// TwinCAT 3 PLC project PLC
// ProgramVersion: 3.1.4022.7
// libraries:
//   Tc2_Standard, * (Beckhoff Automation GmbH)
//   Tc2_System, * (Beckhoff Automation GmbH)
//   Tc2_Utilities, * (Beckhoff Automation GmbH)
//   Tc3_Module, * (Beckhoff Automation GmbH)
//   TcUnit, * (www.tcunit.org)
// project tree:
//   Behavioral Patterns/Command/ I_Command.TcIO, NoCommand.TcPOU
//   Behavioral Patterns/Observer/ Class Diagram Observer.TcCD (not stored), Observable.TcPOU, I_Observable.TcIO, I_Observer.TcIO
//   Behavioral Patterns/Singleton/ I_Singleton.TcIO, Singleton.TcPOU, MySingleton.TcPOU
//   Test/Behavioral Patterns/Singleton/ SingletonPatternTest.TcPOU
//   UseCase/Behavioral Patterns/Command/Clients %28Receivers%29/ Gate.TcPOU (not stored), Light.TcPOU (not stored)
//   UseCase/Behavioral Patterns/Command/Commands/ I_OffCommand.TcIO, I_CloseCommand.TcIO, I_OnCommand.TcIO, I_OpenCommand.TcIO, OffCommand.TcPOU, CloseCommand.TcPOU, OnCommand.TcPOU, OpenCommand.TcPOU
//   UseCase/Behavioral Patterns/Command/Invokers/ Tp10.TcPOU
//   UseCase/Behavioral Patterns/Command/ P_CommandPattern.TcPOU
//   UseCase/Behavioral Patterns/Decorator/ P_Decorator.TcPOU
//   UseCase/Behavioral Patterns/Decorator/StringBuilder/ StringBuilder.TcPOU
//   UseCase/Behavioral Patterns/Singleton/ P_Singleton.TcPOU
//   UseCase/Behavioral Patterns/Singleton/SingletonByProxy1/ P_SingletonByProxy.TcPOU, ProxyToSingleton.TcPOU, Proxy_Interface.TcIO, RealSingleton.TcPOU
//   UseCase/Behavioral Patterns/Singleton/SingletonByProxy/ I_MessageLogger.TcIO, MessageLogger.TcPOU, MessageLoggerSingleton.TcPOU
//   _Interfaces/ I_CyclicCall.TcIO
//   / MAIN.TcPOU, Param.TcGVL, PlcTask.TcTTO
//   Test/Behavioral Patterns/Observer/ ObserverPatternTest.TcPOU
//   Test/ P_TEST.TcPOU
//   UseCase/Behavioral Patterns/Observer/ EventPublisherWithInheritance.TcPOU, EventPublisherWithoutInheritance.TcPOU, FB_EventSubscriber.TcPOU, FB_EventSubscriber2.TcPOU, I_EventPublisher.TcIO, P_ObserverPattern.TcPOU, _Class Diagram Observer Use Case.TcCD (not stored)
//   UseCase/ P_USE_CASES.TcPOU
// real-time tasks:
//   TASK PlcTask: cycle T#10ms, priority 20, ADS port 350

CONFIGURATION PLC
    RESOURCE PLC ON TwinCAT3
        TASK PlcTask(INTERVAL := T#10ms, PRIORITY := 20);
        PROGRAM MAIN WITH PlcTask : MAIN;
    END_RESOURCE
END_CONFIGURATION

// ---- Param.TcGVL
{attribute 'qualified_only'}
VAR_GLOBAL CONSTANT
	MaxObservers 	: INT := 5;	
END_VAR

// ---- Behavioral Patterns/Command/I_Command.TcIO
INTERFACE I_Command

METHOD Execute
VAR_INPUT
END_VAR
END_METHOD

END_INTERFACE

// ---- Behavioral Patterns/Observer/I_Observable.TcIO
INTERFACE I_Observable

METHOD Attach : bool
VAR_INPUT
	observer			: I_Observer;
END_VAR
END_METHOD

METHOD Detach : BOOL
VAR_INPUT
	observer			: I_Observer;
END_VAR
END_METHOD

END_INTERFACE

// ---- Behavioral Patterns/Observer/I_Observer.TcIO
INTERFACE I_Observer

METHOD Update : BOOL
VAR_INPUT
END_VAR
END_METHOD

END_INTERFACE

// ---- Behavioral Patterns/Singleton/I_Singleton.TcIO
INTERFACE I_Singleton

METHOD Message : String
VAR_INPUT
END_VAR
END_METHOD

END_INTERFACE

// ---- UseCase/Behavioral Patterns/Command/Commands/I_OffCommand.TcIO
INTERFACE I_OffCommand

PROPERTY IsOff : Bool
GET
END_GET
END_PROPERTY

METHOD Off
END_METHOD

END_INTERFACE

// ---- UseCase/Behavioral Patterns/Command/Commands/I_CloseCommand.TcIO
INTERFACE I_CloseCommand

METHOD Close
END_METHOD

PROPERTY IsClosed : Bool
GET
END_GET
END_PROPERTY

END_INTERFACE

// ---- UseCase/Behavioral Patterns/Command/Commands/I_OnCommand.TcIO
INTERFACE I_OnCommand

PROPERTY IsOn : Bool
GET
END_GET
END_PROPERTY

METHOD On
END_METHOD

END_INTERFACE

// ---- UseCase/Behavioral Patterns/Command/Commands/I_OpenCommand.TcIO
INTERFACE I_OpenCommand

PROPERTY IsOpen : Bool
GET
END_GET
END_PROPERTY

METHOD Open
END_METHOD

END_INTERFACE

// ---- UseCase/Behavioral Patterns/Singleton/SingletonByProxy1/Proxy_Interface.TcIO
INTERFACE Proxy_Interface

///Illustrative method of the pattern
METHOD Set_Background
VAR_INPUT
	///HEX value to be set as background color
	newBackground: DWORD;
END_VAR
END_METHOD

END_INTERFACE

// ---- UseCase/Behavioral Patterns/Singleton/SingletonByProxy/I_MessageLogger.TcIO
INTERFACE I_MessageLogger

METHOD LogMessage : String
VAR_INPUT
	Message			: STRING;
END_VAR
END_METHOD

PROPERTY message : string
GET
END_GET
END_PROPERTY

END_INTERFACE

// ---- _Interfaces/I_CyclicCall.TcIO
INTERFACE I_CyclicCall

METHOD CyclicCall
END_METHOD

END_INTERFACE

// ---- UseCase/Behavioral Patterns/Observer/I_EventPublisher.TcIO
INTERFACE I_EventPublisher EXTENDS I_Observable

PROPERTY Event : int
GET
END_GET
END_PROPERTY

END_INTERFACE

// ---- MAIN.TcPOU
PROGRAM MAIN
VAR
// *************** ROUTER
	// router info (memory consumption)
	fbGetRouterStatusInfo 	: FB_GetRouterStatusInfo;
	stTCRouterStatusInfo	: ST_TCRouterStatusInfo;
	memAvailable			: DWORD;
END_VAR

// TcUnit tests
P_TEST();

// Use cases implementations
P_USE_CASES();

// *************** ROUTER INFO
// router status
fbGetRouterStatusInfo(
	sNetId:= , 
	bExecute:= NOT fbGetRouterStatusInfo.bBusy, 
	tTimeout:= , 
	bBusy=> , 
	bError=> , 
	nErrID=> , 
	info=> stTCRouterStatusInfo
	);
IF stTCRouterStatusInfo.maxMemAvail	> 0 THEN
	memAvailable := stTCRouterStatusInfo.maxMemAvail;
END_IF

END_PROGRAM

// ---- Test/P_TEST.TcPOU
PROGRAM P_TEST
VAR
	fbObserver_Pattern_Test					: ObserverPatternTest;
	fbSingleton_Pattern_Test				: SingletonPatternTest;
END_VAR

tcUnit.RUN();

END_PROGRAM

// ---- Test/Behavioral Patterns/Observer/ObserverPatternTest.TcPOU
FUNCTION_BLOCK ObserverPatternTest EXTENDS tcUnit.FB_TestSuite
VAR
	// Unit test use the implementation of the use case so both 
	// base blocks and use case blocks are tested at once
	eventPublisher					: EventPublisherWithInheritance;
	//eventSubscriber					: ARRAY[1..param.MaxObservers+1] OF FB_EventSubscriber[(eventPublisher),(eventPublisher),(0),(0),(0),(0)];	// Max + 1 for unit test	// Pass the interface reference to the instances is not possible?	
	eventSubscriber					: ARRAY[1..param.MaxObservers+1] OF FB_EventSubscriber(0);	// Max + 1 for unit test	// Pass the interface reference to the instances is not possible?	
END_VAR

ObservableAttachesAnObserver();
ObservableAttachesASecondObserver();
ObservableAttachesTooMuchObservers();
ObserverFetchesCorrectData();

METHOD ObservableAttachesAnObserver
TEST('ObservableAttachesAnObserver');

// pass observee to subscriber
eventSubscriber[1].ChangePublisher(eventPublisher);

// First loop attaches the observer to the observee 
eventSubscriber[1].CyclicCall();

// One subscriber should be attached
AssertEquals_INT(
	Expected	:= 1, 
	Actual		:= eventPublisher.NoOfAttachedObservers, 
	Message 	:= 'Attaching a subscriber failed'
	);
	
TEST_FINISHED();
END_METHOD

METHOD ObservableAttachesASecondObserver
TEST('ObservableAttachesASecondObserver');

// pass observee to subscriber
eventSubscriber[2].ChangePublisher(eventPublisher);

// First loop attaches another observer to the observee 
eventSubscriber[2].CyclicCall();

// One extra subscriber should be attached
AssertEquals_INT(
	Expected	:= 2, 
	Actual		:= eventPublisher.NoOfAttachedObservers, 
	Message 	:= 'Attaching a second subscriber failed'
	);
	
TEST_FINISHED();
END_METHOD

METHOD ObservableAttachesTooMuchObservers
VAR
	i						: INT;
END_VAR
TEST('ObservableAttachesTooMuchObservers');

// First loop attaches another observer to the observee 
FOR i := 3 TO Param.MaxObservers + 1 DO
	// pass observee to subscriber
	eventSubscriber[i].ChangePublisher(eventPublisher);
	eventSubscriber[i].CyclicCall();
END_FOR
	
// Max no of subscribers should be attached
AssertEquals_INT(
	Expected	:= Param.MaxObservers, 
	Actual		:= eventPublisher.NoOfAttachedObservers, 
	Message 	:= 'Too many subscribers were registered'
	);
	
TEST_FINISHED();
END_METHOD

// Tests the complete observer pattern flow
METHOD ObserverFetchesCorrectData
VAR
	message					: T_MaxString;
	fbFormatString			: FB_FormatString;
	i: INT;
END_VAR
TEST('ObserverFetchesCorrectData');

// Change the event in the publisher (in the example it is an INT) 
eventPublisher.ChangeEvent := eventPublisher.Event + 1;
eventPublisher.CyclicCall();

FOR i := 1 TO Param.MaxObservers DO
	fbFormatString(sFormat:= 'Observer %d did not receive the correct data', arg1:= F_INT(i), sOut=> message);
	AssertEquals_INT(1 , eventSubscriber[i].event, message);
END_FOR

TEST_FINISHED();
END_METHOD

END_FUNCTION_BLOCK

// ---- UseCase/Behavioral Patterns/Observer/EventPublisherWithInheritance.TcPOU
{attribute 'no_explicit_call' := 'FB_EventPublisher is a CLASS and must be accessed using methods or properties'}
FUNCTION_BLOCK EventPublisherWithInheritance EXTENDS Observable IMPLEMENTS I_CyclicCall, I_EventPublisher
VAR
	_event							: INT;
	eventPrev						: INT;
END_VAR


// The body of a class must not be used for code.  
// Cyclic code should be called from a method if needed.

PROPERTY PUBLIC ChangeEvent : int
SET
// IMPLEMENTED ONLY FOR TESTING PURPOSES
VAR
END_VAR
_event := changeEvent;
END_SET
END_PROPERTY

METHOD CyclicCall
IF eventPrev <> _event 			THEN
	notify();
	eventPrev := _event;
END_IF
END_METHOD

// IMPLEMENTED ONLY FOR TESTING PURPOSES
PROPERTY Event : int
GET
event := _event;
END_GET
END_PROPERTY

END_FUNCTION_BLOCK

// ---- Behavioral Patterns/Observer/Observable.TcPOU
{attribute 'no_explicit_call' := 'Observable is a CLASS and must be accessed using methods or properties'}
FUNCTION_BLOCK Observable IMPLEMENTS I_Observable
VAR
	verbose							: BOOL := TRUE;
	// Make sure the list of references to subscribers is updated after online change 
	observers						: ARRAY[1..param.MaxObservers] OF I_Observer;
END_VAR


// The body of a class must not be used for code.  
// Cyclic code should be called from a method if needed.

METHOD Attach : BOOL
VAR_INPUT
	observer			: I_Observer;
END_VAR
VAR
	i					: INT;
END_VAR
(* default *)
attach := FALSE;

(* loop if the subscriber is already registered *)
FOR i := 1 TO param.MaxObservers DO
	IF observers[i] = observer 	THEN
		observer.update();
		attach := TRUE;
		RETURN;
	END_IF
END_FOR

(* loop for first free position if not yet attached *)
FOR i := 1 TO param.MaxObservers DO
	IF observers[i] = 0 	THEN
		observers[i] := observer;
		message('Observer registered');
		observer.update();
		attach := TRUE;
		EXIT;
	END_IF
END_FOR
END_METHOD

METHOD Detach : BOOL
VAR_INPUT
	observer			: I_Observer;
END_VAR
VAR
	i					: INT;
END_VAR
(* default *)
detach := FALSE;

(* loop if the subscriber is already registered *)
FOR i := 1 TO param.MaxObservers DO
	IF observers[i] = observer 	THEN
		observers[i] := 0;
		message('Observer deregistered');
		detach := TRUE;
		RETURN;
	END_IF
END_FOR
END_METHOD

{attribute 'call_after_online_change_slot' := '0'}
METHOD PRIVATE fbreinit
(*	!!!!!!!!!!!!!!!!!!!!!!!!!!!!!!!!!
   	THIS METHOD is force called after every online change 
   	!= the fb_reinit system call that will be called after the instance of the concerned function block has been copied 
 	(during an online change after modifications in the function block declaration)

	This is necessary since both observer en observee have references to one other
	!!!!!!!!!!!!!!!!!!!!!!!!!!!!!!!!!	*) 
VAR
	i					: INT;
END_VAR
(* loop if the subscriber is already registered *)
FOR i := 1 TO param.MaxObservers DO
	observers[i] := 0;
END_FOR
breinit:=NOT breinit; // flip the test marker
END_METHOD

METHOD PRIVATE Message : BOOL
VAR_INPUT
	strArg						: STRING;
END_VAR
// Log message
IF verbose  THEN
	ADSLOGSTR(
		msgCtrlMask := ADSLOG_MSGTYPE_HINT OR ADSLOG_MSGTYPE_LOG, // ADSLOG_MSGTYPE_ERROR OR ADSLOG_MSGTYPE_LOG, 
		msgFmtStr 	:= '%s',
		strArg 		:= strArg
		);
END_IF
END_METHOD

PROPERTY NoOfAttachedObservers : int
GET
VAR
	i							: INT;
END_VAR
// In stead of using an internal counter that could fail
// run through the array of attached observers
(* loop for first free position if not yet attached *)
NoOfAttachedObservers := 0;
FOR i := 1 TO param.MaxObservers DO
	IF observers[i] <> 0 	THEN
		NoOfAttachedObservers := NoOfAttachedObservers + 1;
	END_IF
END_FOR
END_GET
END_PROPERTY

METHOD Notify : BOOL
VAR
	i			: INT;
END_VAR
(* default *)
notify := FALSE;

(* loop if the subscriber is already registered *)
FOR i := 1 TO param.MaxObservers DO
	IF observers[i] <> 0 	THEN
		observers[i].update();
	END_IF
END_FOR
END_METHOD

END_FUNCTION_BLOCK

// ---- UseCase/Behavioral Patterns/Observer/FB_EventSubscriber.TcPOU
{attribute 'no_explicit_call' := 'FB_EventSubscriber is a CLASS and must be accessed using methods or properties'}
FUNCTION_BLOCK FB_EventSubscriber IMPLEMENTS I_CyclicCall, I_Observer
VAR	
	_eventPublisher					: I_EventPublisher;
	_event							: INT;
	
	verbose							: BOOL := TRUE;

	// Register after online change 
	registeredAtPublisher			: BOOL;	
	
	
	arr				: ARRAY[0..100] OF BOOL;
END_VAR


// The body of a class must not be used for code.  
// Cyclic code should be called from a method if needed.

METHOD ChangePublisher
VAR_INPUT
	eventPublisher					: I_EventPublisher;
END_VAR
_eventPublisher := eventPublisher;
END_METHOD

METHOD CyclicCall
// Did we already register in the publisher?
IF NOT registeredAtPublisher	THEN
	registeredAtPublisher := _eventPublisher.attach(THIS^);
END_IF
END_METHOD

// IMPLEMENTED ONLY FOR TESTING PURPOSES
PROPERTY Event : int
GET
event := _event;
END_GET
END_PROPERTY

METHOD FB_init : BOOL
VAR_INPUT
	bInitRetains	 				: BOOL; // if TRUE, the retain variables are initialized (warm start / cold start)
	bInCopyCode 					: BOOL;  // if TRUE, the instance afterwards gets moved into the copy code (online change)
	EventPublisher					: I_EventPublisher;
END_VAR
_eventPublisher := eventPublisher;
END_METHOD

{attribute 'call_after_online_change_slot' := '0'}
METHOD PRIVATE fbreinit

(*	!!!!!!!!!!!!!!!!!!!!!!!!!!!!!!!!!
   	THIS METHOD is force called after every online change 
   	!= the fb_reinit system call that will be called after the instance of the concerned function block has been copied 
 	(during an online change after modifications in the function block declaration)

	This is necessary since both observer en observee have references to one other
	!!!!!!!!!!!!!!!!!!!!!!!!!!!!!!!!!	*)
registeredAtPublisher := FALSE;
breinit:=not breinit; // flip the test marker
END_METHOD

METHOD PRIVATE Message : BOOL
VAR_INPUT
	dintArg						: DINT;
END_VAR
// Log message
IF verbose  THEN
	ADSLOGDINT(
		msgCtrlMask := ADSLOG_MSGTYPE_HINT OR ADSLOG_MSGTYPE_LOG, // ADSLOG_MSGTYPE_ERROR OR ADSLOG_MSGTYPE_LOG, 
		msgFmtStr 	:= 'Subscriber 1 knows the value changed to %d',
		dintArg 	:= dintArg
		);
END_IF
END_METHOD

METHOD Update : BOOL
// the publisher mentions an update, fetch the data
_event := _eventPublisher.event;
message(TO_DINT(_event));
END_METHOD

END_FUNCTION_BLOCK

// ---- Test/Behavioral Patterns/Singleton/SingletonPatternTest.TcPOU
FUNCTION_BLOCK SingletonPatternTest EXTENDS tcUnit.FB_TestSuite
VAR
	messageLogger1				: MessageLogger;
	messageLogger2				: MessageLogger;
	messageLogger3				: MessageLogger;
	myMessage1					: STRING := 'Message 1';
	myMessage2					: STRING := 'Message 2';
	myMessage3					: STRING := 'Message 3';
END_VAR

SendMessageToMessageLogger1();
SendMessageToMessageLogger2();
SendMessageToMessageLogger3();

METHOD SendMessageToMessageLogger1
TEST('SendMessageToMessageLogger1');

// Log 'message 1' to the first messagelogger instance
messageLogger1.LogMessage(myMessage1);

// The message should be available in the first messagelogger
AssertEquals_STRING(
	Expected	:= myMessage1, 
	Actual		:= messageLogger1.message, 
	Message 	:= 'Message1 was not received by message logger 1'
	);
	
TEST_FINISHED();
END_METHOD

METHOD SendMessageToMessageLogger2
TEST('SendMessageToMessageLogger2');

// Log 'message 2' to a second messagelogger instance
messageLogger2.LogMessage(myMessage2);

// The message should be available in the second messagelogger
AssertEquals_STRING(
	Expected	:= myMessage2, 
	Actual		:= messageLogger2.message, 
	Message 	:= 'Message2 was not received by message logger 2'
	);
	
// Since there is already an instance of the singleton, also message logger 1 should have received message 2
AssertEquals_STRING(
	Expected	:= 'Message 2', 
	Actual		:= messageLogger1.message, 
	Message 	:= 'Message2 was not received by message logger 1'
	);
		
TEST_FINISHED();
END_METHOD

METHOD SendMessageToMessageLogger3
VAR_INPUT
END_VAR
TEST('SendMessageToMessageLogger3');

// Log 'message 2' to a second messagelogger instance
messageLogger3.LogMessage(myMessage3);

// The message should be available in the second messagelogger
AssertEquals_STRING(
	Expected	:= myMessage3, 
	Actual		:= messageLogger3.message, 
	Message 	:= 'Message3 was not received by message logger 3'
	);
	
// Since there is already an instance of the singleton, also message logger 1 should have received message 2
AssertEquals_STRING(
	Expected	:= myMessage3, 
	Actual		:= messageLogger1.message, 
	Message 	:= 'Message3 was not received by message logger 1'
	);
		
TEST_FINISHED();
END_METHOD

END_FUNCTION_BLOCK

// ---- UseCase/Behavioral Patterns/Singleton/SingletonByProxy/MessageLogger.TcPOU
{attribute 'no_explicit_call' := 'MySingleton is a CLASS and must be accessed using methods or properties'}
FUNCTION_BLOCK MessageLogger IMPLEMENTS I_MessageLogger
VAR_STAT 	// VAR_STAT makes sure all new instances use the same initialized vars
	messageLogger					: I_MessageLogger;				
	messageLoggerSingleton			: POINTER TO MessageLoggerSingleton;
END_VAR

METHOD FB_exit : BOOL
VAR_INPUT
	bInCopyCode : BOOL; // if TRUE, the exit method is called for exiting an instance that is copied afterwards (online change).
END_VAR
// Delete the dynamic instance at FB_exit 
IF messageLoggerSingleton <> 0	THEN
	messageLogger := 0;					// Clear interface
	__DELETE(messageLoggerSingleton);	// Delete the instance
	messageLoggerSingleton:=0;			// Clear the pointer
END_IF
END_METHOD

METHOD FB_init : BOOL
VAR_INPUT
	bInitRetains : BOOL; // if TRUE, the retain variables are initialized (warm start / cold start)
	bInCopyCode : BOOL;  // if TRUE, the instance afterwards gets moved into the copy code (online change)
END_VAR
// first instance? 
IF messageLoggerSingleton = 0	THEN
	messageLoggerSingleton := __NEW(messageLoggerSingleton);
	messageLogger := messageLoggerSingleton^;
END_IF
END_METHOD

METHOD LogMessage : STRING
VAR_INPUT
	message			: STRING;
END_VAR
IF messageLogger <> 0 THEN
	messageLogger.LogMessage(message);
END_IF
END_METHOD

{warning 'add property implementation'}
PROPERTY message : STRING
GET
message := messageLogger.message;
END_GET
END_PROPERTY

END_FUNCTION_BLOCK

// ---- Behavioral Patterns/Singleton/MySingleton.TcPOU
{attribute 'no_explicit_call' := 'MySingleton is a CLASS and must be accessed using methods or properties'}
FUNCTION_BLOCK MySingleton IMPLEMENTS I_Singleton
VAR 
	singleton					: I_Singleton;	// define the static class instance	
	singletonInstance			: POINTER TO Singleton;
END_VAR

METHOD FB_exit : BOOL
VAR_INPUT
	bInCopyCode : BOOL; // if TRUE, the exit method is called for exiting an instance that is copied afterwards (online change).
END_VAR
// first instance? 
IF singletonInstance <> 0	THEN
	singleton := 0;
	__DELETE(singletonInstance);
	singletonInstance:=0;
END_IF
END_METHOD

METHOD FB_init : BOOL
VAR_INPUT
	bInitRetains : BOOL; // if TRUE, the retain variables are initialized (warm start / cold start)
	bInCopyCode : BOOL;  // if TRUE, the instance afterwards gets moved into the copy code (online change)
END_VAR
// first instance? 
IF singletonInstance = 0	THEN
	singletonInstance := __NEW(Singleton);
	singleton := singletonInstance^;
END_IF
END_METHOD

METHOD FB_reinit : BOOL
VAR_INPUT
END_VAR
__DELETE(singletonInstance);
singleton := 0;
END_METHOD

METHOD Message : STRING
IF singleton <> 0 THEN
	Message := singleton.Message();
END_IF
END_METHOD

END_FUNCTION_BLOCK

// ---- Behavioral Patterns/Singleton/Singleton.TcPOU
{attribute 'enable_dynamic_creation'}
{attribute 'no_explicit_call' := 'Singleton is a CLASS and must be accessed using methods or properties'}
FUNCTION_BLOCK Singleton IMPLEMENTS I_Singleton

METHOD Message : STRING
Message := 'myMessage';
END_METHOD

END_FUNCTION_BLOCK

// ---- UseCase/Behavioral Patterns/Singleton/SingletonByProxy/MessageLoggerSingleton.TcPOU
{attribute 'enable_dynamic_creation'}
{attribute 'no_explicit_call' := 'Singleton is a CLASS and must be accessed using methods or properties'}
FUNCTION_BLOCK MessageLoggerSingleton IMPLEMENTS I_MessageLogger // USE MessageLogger!!
VAR
	_message			: STRING;
END_VAR

METHOD LogMessage : STRING
VAR_INPUT
	message			: STRING;
END_VAR
_message := message;
END_METHOD

{warning 'add property implementation'}
PROPERTY message : STRING
GET
message  := _message;
END_GET
END_PROPERTY

END_FUNCTION_BLOCK

// ---- UseCase/P_USE_CASES.TcPOU
PROGRAM P_USE_CASES
VAR
END_VAR

// Behavioral patterns
P_ObserverPattern();
P_Decorator();
P_CommandPattern();
P_Singleton();
//P_SingletonByProxy();

END_PROGRAM

// ---- UseCase/Behavioral Patterns/Observer/P_ObserverPattern.TcPOU
PROGRAM P_ObserverPattern
VAR
	eventPublisher					: EventPublisherWithInheritance;
	eventPublisher2					: EventPublisherWithoutInheritance;	
	
	eventSubscriber					: FB_EventSubscriber(eventPublisher);	
	eventSubscriber2				: FB_EventSubscriber2(eventPublisher2);	
	
	refEventSubscriber				: REFERENCE TO FB_EventSubscriber := eventSubscriber;
	refEventSubscriber2				: REFERENCE TO FB_EventSubscriber2 := eventSubscriber2;	
	
	triggerEvent					: BOOL;
END_VAR

// Property changeEvent was only to be able to change the event from outside for the unit test
// Change according the use case of the observer
IF triggerEvent	THEN
	eventPublisher.changeEvent := eventPublisher.event + 1;
	eventPublisher2.changeEvent := eventPublisher2.event + 1;
	triggerEvent := FALSE;
END_IF
eventPublisher.CyclicCall();
eventPublisher2.CyclicCall();

eventSubscriber.CyclicCall();
eventSubscriber2.CyclicCall();

END_PROGRAM

// ---- UseCase/Behavioral Patterns/Observer/EventPublisherWithoutInheritance.TcPOU
{attribute 'no_explicit_call' := 'FB_EventPublisher is a CLASS and must be accessed using methods or properties'}
FUNCTION_BLOCK EventPublisherWithoutInheritance IMPLEMENTS I_CyclicCall, I_EventPublisher
VAR
	_event							: INT;
	eventPrev						: INT;
	
	observable						: Observable;
END_VAR


// The body of a class must not be used for code.  
// Cyclic code should be called from a method if needed.

METHOD Attach : BOOL
VAR_INPUT
	observer	: I_Observer;
END_VAR
Attach := observable.Attach(observer);
END_METHOD

PROPERTY PUBLIC ChangeEvent : int
SET
// IMPLEMENTED ONLY FOR TESTING PURPOSES
VAR
END_VAR
_event := changeEvent;
END_SET
END_PROPERTY

METHOD CyclicCall
IF eventPrev <> _event 			THEN
	observable.Notify();
	eventPrev := _event;
END_IF
END_METHOD

METHOD Detach : BOOL
VAR_INPUT
	observer	: I_Observer;
END_VAR
Detach := observable.Detach(observer);
END_METHOD

// IMPLEMENTED ONLY FOR TESTING PURPOSES
PROPERTY Event : int
GET
event := _event;
END_GET
END_PROPERTY

END_FUNCTION_BLOCK

// ---- UseCase/Behavioral Patterns/Observer/FB_EventSubscriber2.TcPOU
{attribute 'no_explicit_call' := 'FB_EventSubscriber2 is a CLASS and must be accessed using methods or properties'}
FUNCTION_BLOCK FB_EventSubscriber2 IMPLEMENTS I_CyclicCall, I_Observer
VAR	
	_eventPublisher					: I_EventPublisher;
	_event							: INT;
	
	verbose							: BOOL := TRUE;

	// Register after online change 
	registeredAtPublisher			: BOOL;
END_VAR

METHOD ChangePublisher
VAR_INPUT
	eventPublisher					: I_EventPublisher;
END_VAR
_eventPublisher := eventPublisher;
END_METHOD

METHOD CyclicCall
// Did we already register in the publisher?
IF NOT registeredAtPublisher	THEN
	registeredAtPublisher := _eventPublisher.attach(THIS^);
END_IF
END_METHOD

// IMPLEMENTED ONLY FOR TESTING PURPOSES
PROPERTY Event : int
GET
event := _event;
END_GET
END_PROPERTY

METHOD FB_init : BOOL
VAR_INPUT
	bInitRetains	 				: BOOL; // if TRUE, the retain variables are initialized (warm start / cold start)
	bInCopyCode 					: BOOL;  // if TRUE, the instance afterwards gets moved into the copy code (online change)
	eventPublisher					: I_EventPublisher;
END_VAR
_eventPublisher := eventPublisher;
END_METHOD

{attribute 'call_after_online_change_slot' := '0'}
METHOD PRIVATE fbreinit

(*	!!!!!!!!!!!!!!!!!!!!!!!!!!!!!!!!!
   	THIS METHOD is force called after every online change 
   	!= the fb_reinit system call that will be called after the instance of the concerned function block has been copied 
 	(during an online change after modifications in the function block declaration)

	This is necessary since both observer en observee have references to one other
	!!!!!!!!!!!!!!!!!!!!!!!!!!!!!!!!!	*)
registeredAtPublisher := FALSE;
breinit:=not breinit; // flip the test marker
END_METHOD

METHOD PRIVATE Message : BOOL
VAR_INPUT
	dintArg						: DINT;
END_VAR
// Log message
IF verbose  THEN
	ADSLOGDINT(
		msgCtrlMask := ADSLOG_MSGTYPE_HINT OR ADSLOG_MSGTYPE_LOG, // ADSLOG_MSGTYPE_ERROR OR ADSLOG_MSGTYPE_LOG, 
		msgFmtStr 	:= 'Subscriber 2 knows the value changed to %d',
		dintArg 	:= dintArg
		);
END_IF
END_METHOD

METHOD Update : BOOL
// the publisher mentions an update, fetch the data
_event := _eventPublisher.event;
message(TO_DINT(_event));
END_METHOD

END_FUNCTION_BLOCK

// ---- UseCase/Behavioral Patterns/Decorator/P_Decorator.TcPOU
PROGRAM P_Decorator
VAR
	ErrorString				: STRING;
	stringBuilder			: StringBuilder;
	ErrorNumber				: INT := 1;
	ErrorMessage			: STRING := 'This is my error message';
END_VAR

ErrorString := stringBuilder
					.Clear()
					.Append('Error number: ')
					.Append(INT_TO_STRING(ErrorNumber))
					.Append('. Message: ')
					.Append(ErrorMessage)
					.Append('.')
					.ToString();

END_PROGRAM

// ---- UseCase/Behavioral Patterns/Decorator/StringBuilder/StringBuilder.TcPOU
(*~
<docu>
	<summary>
			Allows to concat strings using fluent interface. It's similar to C# StringBuilder class
			Usage as follows :
			<code>
				ErrorString := _stringBuilder
					.Clear()
					.Append('Error number: ')
					.Append(INT_TO_STRING(ErrorNumber))
					.Append('. Message: ')
					.Append(ErrorMessage)
					.Append('.')
					.ToString();
			</code>
			
			Inspired by Gerhard Barteling blogpost at https://www.plccoder.com/fluent-code/
	</summary>				
</docu>	
~*)	
FUNCTION_BLOCK StringBuilder
VAR
	{attribute 'hide'}
    _workString:STRING(255);
END_VAR

(*
	Thanks to https://github.com/bengeisler/TcLog
*)

METHOD PROTECTED AnyToString : STRING(255)
VAR_INPUT
	Data:	ANY;
END_VAR
VAR
	pAnyBOOL		: POINTER TO BOOL; 
	pAnyBYTE		: POINTER TO BYTE; 
	pAnyWORD		: POINTER TO WORD; 
	pAnyDWORD		: POINTER TO DWORD;
	pAnyLWORD		: POINTER TO LWORD;
	pAnySINT		: POINTER TO SINT; 
	pAnyUSINT		: POINTER TO USINT;
	pAnyINT			: POINTER TO INT;  
	pAnyUINT		: POINTER TO UINT; 
	pAnyDINT		: POINTER TO DINT; 
	pAnyUDINT		: POINTER TO UDINT;
	pAnyLINT		: POINTER TO LINT; 
	pAnyULINT		: POINTER TO ULINT;
	pAnyLTIME		: POINTER TO LTIME;	
	pAnyReal 		: POINTER TO REAL;
	pAnyLReal		: POINTER TO LREAL;	
	pAnyDateAndTime : POINTER TO DATE_AND_TIME;
	pAnyDate		: POINTER TO DATE;
	pAnyTime		: POINTER TO TIME;
	pAnyWString		: POINTER TO WSTRING;
	pAnyTOD			: POINTER TO TOD;
	pAnyString		: POINTER TO STRING;	
	sString			: T_MAXSTRING;
	wWString		: WSTRING;
END_VAR
IF Data.TypeClass = __SYSTEM.TYPE_CLASS.TYPE_REAL THEN
	pAnyReal := Data.pValue;
	AnyToString := REAL_TO_STRING(pAnyReal^);
	
ELSIF Data.TypeClass = __SYSTEM.TYPE_CLASS.TYPE_LREAL THEN
	pAnyLReal := Data.pValue;
	AnyToString := LREAL_TO_STRING(pAnyLReal^);
	
ELSIF Data.TypeClass = __SYSTEM.TYPE_CLASS.TYPE_DATEANDTIME THEN
	pAnyDateAndTime := Data.pValue;
	AnyToString := DT_TO_STRING(pAnyDateAndTime^);	
	
ELSIF Data.TypeClass = __SYSTEM.TYPE_CLASS.TYPE_DATE THEN
	pAnyDate := Data.pValue;
	AnyToString := DATE_TO_STRING(pAnyDate^);
	
ELSIF Data.TypeClass = __SYSTEM.TYPE_CLASS.TYPE_TIME THEN
	pAnyTime := Data.pValue;
	AnyToString := TIME_TO_STRING(pAnyTime^);
	
ELSIF Data.TypeClass = __SYSTEM.TYPE_CLASS.TYPE_STRING THEN
	pAnyString := Data.pValue;
	AnyToString := pAnyString^;
	
ELSIF Data.TypeClass = __SYSTEM.TYPE_CLASS.TYPE_WSTRING THEN
	pAnyWString := Data.pValue;
	wWString := pAnyWString^;
	WSTRING_TO_STRING2(ADR(sString), ADR(wWstring), SIZEOF(wWString));
	AnyToString := sString;
	
ELSIF Data.TypeClass = __SYSTEM.TYPE_CLASS.TYPE_TIMEOFDAY THEN
	pAnyTOD := Data.pValue;
	AnyToString := TOD_TO_STRING(pAnyTOD^);
ELSIF Data.TypeClass = __SYSTEM.TYPE_CLASS.TYPE_BOOL THEN 	
	pAnyBOOL := Data.pValue;
	AnyToString := BOOL_TO_STRING(pAnyBool^);
ELSIF Data.TypeClass = __SYSTEM.TYPE_CLASS.TYPE_BYTE THEN
	pAnyBYTE := Data.pValue;
	AnyToString := BYTE_TO_STRING(pAnyBYTE^);	
ELSIF Data.TypeClass = __SYSTEM.TYPE_CLASS.TYPE_WORD THEN
	pAnyWORD := Data.pValue;
	AnyToString := WORD_TO_STRING(pAnyWORD^);	
ELSIF Data.TypeClass = __SYSTEM.TYPE_CLASS.TYPE_DWORD THEN
	pAnyDWORD := Data.pValue;	
	AnyToString := DWORD_TO_STRING(pAnyDWORD^);
ELSIF Data.TypeClass = __SYSTEM.TYPE_CLASS.TYPE_LWORD THEN
	pAnyLWORD := Data.pValue;	
	AnyToString := LWORD_TO_STRING(pAnyLWORD^);
ELSIF Data.TypeClass = __SYSTEM.TYPE_CLASS.TYPE_SINT THEN
	pAnySINT := Data.pValue;	
	AnyToString := SINT_TO_STRING(pAnySINT^);					
ELSIF Data.TypeClass = __SYSTEM.TYPE_CLASS.TYPE_USINT THEN
	pAnyUSINT := Data.pValue;	
	AnyToString := USINT_TO_STRING(pAnyUSINT^);	
ELSIF Data.TypeClass = __SYSTEM.TYPE_CLASS.TYPE_INT THEN
	pAnyINT := Data.pValue;	
	AnyToString := INT_TO_STRING(pAnyINT^);	
ELSIF Data.TypeClass = __SYSTEM.TYPE_CLASS.TYPE_UINT THEN
	pAnyUINT := Data.pValue;	
	AnyToString := UINT_TO_STRING(pAnyUINT^);	
ELSIF Data.TypeClass = __SYSTEM.TYPE_CLASS.TYPE_DINT THEN
	pAnyDINT := Data.pValue;	
	AnyToString := DINT_TO_STRING(pAnyDINT^);	
ELSIF Data.TypeClass = __SYSTEM.TYPE_CLASS.TYPE_UDINT THEN
	pAnyUDINT := Data.pValue;	
	AnyToString := UDINT_TO_STRING(pAnyUDINT^);	
ELSIF Data.TypeClass = __SYSTEM.TYPE_CLASS.TYPE_LINT THEN
	pAnyLINT := Data.pValue;	
	AnyToString := LINT_TO_STRING(pAnyLINT^);	
ELSIF Data.TypeClass = __SYSTEM.TYPE_CLASS.TYPE_ULINT THEN
	pAnyULINT := Data.pValue;	
	AnyToString := ULINT_TO_STRING(pAnyULINT^);	
ELSIF Data.TypeClass = __SYSTEM.TYPE_CLASS.TYPE_LTIME THEN
	pAnyLTIME := Data.pValue;	
	AnyToString := LTIME_TO_STRING(pAnyLTIME^);		
ELSE	
	AnyToString := ANY_TO_STRING(Data.pValue^);
END_IF
END_METHOD

METHOD Append : REFERENCE TO StringBuilder
VAR_INPUT
    Text :STRING(255); 
END_VAR
_workString := Concat(_workString,text);
Append REF= THIS^;
END_METHOD

METHOD INTERNAL AppendAny : REFERENCE TO StringBuilder
VAR_INPUT
	Data : ANY;
END_VAR
_workString := Concat(_workString,AnyToString(Data));
AppendAny REF= THIS^;
END_METHOD

METHOD Clear : REFERENCE TO StringBuilder
_workString := '';
Clear REF= THIS^;
END_METHOD

METHOD ToString : STRING(255)
ToString := _workString;
END_METHOD

END_FUNCTION_BLOCK

// ---- UseCase/Behavioral Patterns/Command/P_CommandPattern.TcPOU
PROGRAM P_CommandPattern
VAR
	lightLivingRoom					: Light;
	lightLivingRoomOnCommand		: OnCommand(OnCommand:=LightLivingRoom);
	lightLivingRoomOffCommand		: OffCommand(OffCommand:=LightLivingRoom);

	lightKitchen					: Light;
	lightKitchenOnCommand			: OnCommand(OnCommand:=LightKitchen);
	lightKitchenOffCommand			: OffCommand(OffCommand:=LightKitchen);

	lightBathroom					: Light;
	lightBathroomOnCommand			: OnCommand(OnCommand:=LightBathroom);
	lightBathroomOffCommand			: OffCommand(OffCommand:=LightBathroom);

	frontGate						: Gate;
	frontGateOpenCommand			: OpenCommand(OpenCommand:=frontGate);
	frontGateCloseCommand			: CloseCommand(CloseCommand:=frontGate);
		
	// TP10 (https://fixsus.be/hardware/tp10)
	tp10MainHallway					: TP10;
	
	init							: BOOL := TRUE;// Initialization	
	
END_VAR

IF init THEN
	// assign the commands to the TP10
	tp10MainHallway.SetCommand(0, lightLivingRoomOnCommand);
	tp10MainHallway.SetCommand(5, lightLivingRoomOffCommand);
	tp10MainHallway.SetCommand(1, lightKitchenOnCommand);
	tp10MainHallway.SetCommand(6, lightKitchenOffCommand);
	tp10MainHallway.SetCommand(2, lightBathroomOnCommand);
	tp10MainHallway.SetCommand(7, lightBathroomOffCommand);
	tp10MainHallway.SetCommand(3, frontGateOpenCommand);
	tp10MainHallway.SetCommand(8, frontGateCloseCommand);
	init := FALSE;
END_IF

// The lights have no cyclic call since they just flip the output

// The gate needs to be processed as long as it is not fully opened or closed after a command
frontGate.CyclicCall();

// Process the tp10's, could be an array of instances that is cyclically called
tp10MainHallway.CyclicCall();

END_PROGRAM

// ---- UseCase/Behavioral Patterns/Command/Commands/OnCommand.TcPOU
{attribute 'no_explicit_call' := 'LightOnCommand is a CLASS and must be accessed using methods or properties'}
FUNCTION_BLOCK OnCommand IMPLEMENTS I_Command
VAR
	_onCommand					: I_OnCommand;
END_VAR


// The body of a class must not be used for code.  
// Cyclic code should be called from a method if needed.

METHOD Execute
_onCommand.On();
END_METHOD

METHOD FB_init : BOOL
VAR_INPUT
	bInitRetains : BOOL; // if TRUE, the retain variables are initialized (warm start / cold start)
	bInCopyCode : BOOL;  // if TRUE, the instance afterwards gets moved into the copy code (online change)
	OnCommand			: I_OnCommand;
END_VAR
_onCommand  := OnCommand;
END_METHOD

END_FUNCTION_BLOCK

// ---- UseCase/Behavioral Patterns/Command/Commands/OffCommand.TcPOU
{attribute 'no_explicit_call' := 'LightOnCommand is a CLASS and must be accessed using methods or properties'}
FUNCTION_BLOCK OffCommand IMPLEMENTS I_Command
VAR
	_offCommand					: I_OffCommand;
END_VAR


// The body of a class must not be used for code.  
// Cyclic code should be called from a method if needed.

METHOD Execute
_offCommand.Off();
END_METHOD

METHOD FB_init : BOOL
VAR_INPUT
	bInitRetains : BOOL; // if TRUE, the retain variables are initialized (warm start / cold start)
	bInCopyCode : BOOL;  // if TRUE, the instance afterwards gets moved into the copy code (online change)
	OffCommand			: I_OffCommand;
END_VAR
_offCommand  := OffCommand;
END_METHOD

END_FUNCTION_BLOCK

// ---- UseCase/Behavioral Patterns/Command/Commands/OpenCommand.TcPOU
{attribute 'no_explicit_call' := 'LightOnCommand is a CLASS and must be accessed using methods or properties'}
FUNCTION_BLOCK OpenCommand IMPLEMENTS I_Command
VAR
	_openCommand					: I_OpenCommand;
END_VAR


// The body of a class must not be used for code.  
// Cyclic code should be called from a method if needed.

METHOD Execute
_openCommand.Open();
END_METHOD

METHOD FB_init : BOOL
VAR_INPUT
	bInitRetains : BOOL; // if TRUE, the retain variables are initialized (warm start / cold start)
	bInCopyCode : BOOL;  // if TRUE, the instance afterwards gets moved into the copy code (online change)
	OpenCommand			: I_OpenCommand;
END_VAR
_openCommand  := OpenCommand;
END_METHOD

END_FUNCTION_BLOCK

// ---- UseCase/Behavioral Patterns/Command/Commands/CloseCommand.TcPOU
{attribute 'no_explicit_call' := 'LightOnCommand is a CLASS and must be accessed using methods or properties'}
FUNCTION_BLOCK CloseCommand IMPLEMENTS I_Command
VAR
	_closeCommand					: I_CloseCommand;
END_VAR


// The body of a class must not be used for code.  
// Cyclic code should be called from a method if needed.

METHOD Execute
_closeCommand.Close();
END_METHOD

METHOD FB_init : BOOL
VAR_INPUT
	bInitRetains : BOOL; // if TRUE, the retain variables are initialized (warm start / cold start)
	bInCopyCode : BOOL;  // if TRUE, the instance afterwards gets moved into the copy code (online change)
	CloseCommand			: I_CloseCommand;
END_VAR
_closeCommand  := CloseCommand;
END_METHOD

END_FUNCTION_BLOCK

// ---- UseCase/Behavioral Patterns/Command/Invokers/Tp10.TcPOU
{attribute 'no_explicit_call' := 'Tp10 is a CLASS and must be accessed using methods or properties'}
FUNCTION_BLOCK Tp10 IMPLEMENTS I_CyclicCall
VAR
	buttons			AT%I*		: ARRAY[0..NOOFCOMMANDS-1] OF BOOL;
	risingTrigger				: ARRAY[0..NOOFCOMMANDS-1] OF R_TRIG;

	commands					: ARRAY[0..NOOFCOMMANDS-1] OF I_Command;
	noCommand					: NoCommand;	// Default command containing NO code in Execute
END_VAR
VAR CONSTANT
	NOOFCOMMANDS				: INT := 10;
END_VAR
/// https://fixsus.be/hardware/tp10


// The body of a class must not be used for code.  
// Cyclic code should be called from a method if needed.

METHOD CyclicCall

VAR
	i: INT;
END_VAR
// Check the pushbuttons
FOR i := 0 TO NOOFCOMMANDS -1 DO
	risingTrigger[i](CLK:=buttons[i]);
	// Issue command if the button was pressed
	IF risingTrigger[i].Q		THEN
		commands[i].Execute();		
	END_IF
END_FOR
END_METHOD

METHOD FB_init : BOOL
VAR_INPUT
	bInitRetains : BOOL; // if TRUE, the retain variables are initialized (warm start / cold start)
	bInCopyCode : BOOL;  // if TRUE, the instance afterwards gets moved into the copy code (online change)
END_VAR
VAR
	i					: INT;
END_VAR
// Initialize the command buttons to NOCommand 
FOR i := 0 TO NOOFCOMMANDS - 1 DO
	Commands[i] := THIS^.noCommand;		// basic initialization of a button, avoids the need of checking for a valid command in the code, just does nothing when pressed
END_FOR
END_METHOD

METHOD RemoveCommand
VAR_INPUT
	slot					: INT;
END_VAR
// Check if the slot no is valid
IF slot >=0 AND slot < NOOFCOMMANDS THEN 
	commands[slot] := noCommand;	
END_IF
END_METHOD

METHOD SetCommand
VAR_INPUT
	slot					: INT;
	command					: I_Command;
END_VAR
// Check if the slot no is valid
IF slot >=0 AND slot < NOOFCOMMANDS THEN 
	commands[slot] := command;	
END_IF
END_METHOD

END_FUNCTION_BLOCK

// ---- Behavioral Patterns/Command/NoCommand.TcPOU
{attribute 'no_explicit_call' := 'NoCommand is a CLASS and must be accessed using methods or properties'}
FUNCTION_BLOCK NoCommand IMPLEMENTS I_Command
VAR
END_VAR
/// Command that does nothing for base initialization

METHOD Execute
END_METHOD

END_FUNCTION_BLOCK

// ---- UseCase/Behavioral Patterns/Singleton/P_Singleton.TcPOU
PROGRAM P_Singleton
VAR
	messageLogger				: MessageLogger;
	messageLogger1				: MessageLogger;
	messageLogger2				: MessageLogger;
	myMessage					: STRING;
	myMessage1					: STRING := 'Message 1';
	myMessage2					: STRING := 'Message 2';
	myMessage3					: STRING := 'Message 3';
END_VAR

// Log 'message 1' to the first messagelogger instance
messageLogger.LogMessage(myMessage1);
myMessage := messageLogger.message;

// Log 'message 2' to a second messagelogger instance
messageLogger1.LogMessage(myMessage2);
myMessage := messageLogger.message;
myMessage := messageLogger1.message;

// Log 'message 3' to a third messagelogger instance
messageLogger2.LogMessage(myMessage3);
myMessage := messageLogger.message;
myMessage := messageLogger2.message;

END_PROGRAM

// ---- UseCase/Behavioral Patterns/Singleton/SingletonByProxy1/P_SingletonByProxy.TcPOU
PROGRAM P_SingletonByProxy
VAR
	///Blue, highly opaque
	dwBlue: DWORD := 16#FF0000FF;
	///Green, highly opaque
	dwGreen: DWORD := 16#FF00FF00;
	///Yellow, highly opaque
	dwYellow: DWORD := 16#FFFFFF00;
	///Creates 3 instances of the ProxyToSingleton class
	instance1: ProxyToSingleton;
	instance2: ProxyToSingleton;
	instance3: ProxyToSingleton;
END_VAR

//The PLC_PRG handles the instanciation of the possible background colours and the ProxyToSingleton instances in order to be used by the Visualization element.
//The viasualization element (The client) handles the request for background change on the RealSingleton object through the ProxyToSinlgeton instances.
//These request are first processed by the ProxyToSingleton object and then passed to the one and only RealSingleton instance.
//The default background colour of the RealSingleton object is 'Blue'

END_PROGRAM

// ---- UseCase/Behavioral Patterns/Singleton/SingletonByProxy1/ProxyToSingleton.TcPOU
///This class is called ProxyToSingleton because it works as a Proxy of the Singleton class. It handles the creation and instanciation of the 
/// RealSingleton class. Something like the proper static method GetInstance(); in any singleton pattern.
///So the ProxyToSingleton class has a static Singleton object as a field and whenever we instanciate a 
/// ProxyToSingleton object we will have the RealSingleton object as its static field .realSingleton^
{attribute 'enable_dynamic_creation' := ''}
FUNCTION_BLOCK ProxyToSingleton IMPLEMENTS Proxy_Interface
VAR_STAT
	///Boolean value to check if there is already a Singleton instance
	bFirstInstance: BOOL := FALSE;
	///Pointer to the first and only instance of the Singleton class
	realSingleton: POINTER TO RealSingleton;
END_VAR

METHOD fb_init
VAR_INPUT
	/// TRUE: the Retain-variables are initialized (reset warm / reset cold)
	bInitRetains: BOOL;
	/// TRUE  the instance will be copied to the copy-code afterward (online change)
	bInCopyCode: BOOL;
END_VAR
//THIS FUNCTION WORKS AS THE CONSTRUCTOR OF THE ProxyToSingleton CLASS
// It handles the creation of the only RealSingleton object. It uses the concept of lazy instanciation.

//If the static property .bFirstInstance is TRUE
IF THIS^.bFirstInstance = TRUE
	
THEN
		//There is already a Singleton object.
		//So we don't have to do anything, this new ProxyToSingleton object will already have the address of the 
		// RealSingleton object in its pointer .realSingleton
	
	ELSE	//If the static property .bFirstInstance is FALSE
	
		//There is not a Singleton object so the ProxyToSingleton object calling the constructor 
		// should create the RealSingleton object in its pointer field .realSingleton 
		//Then we change the status of the static variable bFirstInstance to TRUE and avoid overwriting the realSingleton address.
		//If the Singleton object is destroyed, .bFirstInstance should be set to FALSE again.
		THIS^.bFirstInstance := TRUE;
		
		//Reference the value of the first RealSingleton instance to the FakeSingleton object to save 
		// the address of the real Singleton instance.
		THIS^.realSingleton := __NEW(RealSingleton);
END_IF
END_METHOD

///Illustrative method of the pattern
METHOD Set_Background
VAR_INPUT
	///HEX value to be set as background color
	newBackground: DWORD;
END_VAR
//The ProxyToSingleton object handles the request and send the appropiate reques to the one and only RealSingleton instance
THIS^.realSingleton^.Set_Background(newBackground);
END_METHOD

END_FUNCTION_BLOCK

// ---- UseCase/Behavioral Patterns/Singleton/SingletonByProxy1/RealSingleton.TcPOU
///This class is called RealSingleton because it works as singleton.  
///As long as we only instanciate ProxyToSingleton objects, this class will work as a Singleton class should work.
///The global access point to this class is the field .realSingleton^ in every ProxyToSingleton object.
{attribute 'enable_dynamic_creation' := ''}
FUNCTION_BLOCK RealSingleton IMPLEMENTS Proxy_Interface
VAR
	///Illustrative field of the pattern to store the HEX value for the background colour
	backgroundColour: DWORD;
END_VAR

METHOD fb_init
VAR_INPUT
	/// TRUE: the Retain-variables are initialized (reset warm / reset cold)
	bInitRetains: BOOL;
	/// TRUE  the instance will be copied to the copy-code afterward (online change)
	bInCopyCode: BOOL;
END_VAR
//The default valur for the background is set
THIS^.Set_Background(P_SingletonByProxy.dwBlue);
END_METHOD

///Illustrative method of the pattern
METHOD Set_Background
VAR_INPUT
	///HEX value to be set as background color
	newBackground: DWORD;
END_VAR
//Writes the backgroundColour field to the passed newBackground value
THIS^.backgroundColour := newBackground;
END_METHOD

END_FUNCTION_BLOCK
